FUNCTION IsInRangeInclusive : BOOL
VAR_INPUT
	value : LREAL;
	range : Range;
END_VAR

IsInRangeInclusive := range.Bottom <= value AND value <= range.Top;

END_FUNCTION

(* stored: Version 1.1.0.1, ProductVersion 3.1.4024.15
   POU IsInRangeInclusive: Id {8dd7d775-21b8-05d0-2476-b7ec38ff0002}, SpecialFunc None *)
